// TIA Portal V17 export
// export: Created 2022-03-12T16:05:35.2903502Z, ExportSetting WithDefaults, DisplayName Totally Integrated Automation Portal, DisplayVersion V17, DisplayName TIA Portal Openness, DisplayVersion V17, DisplayName TIA Portal Version Control Interface, DisplayVersion V17, DisplayName STEP 7 Professional, DisplayVersion V17, DisplayName STEP 7 Safety, DisplayVersion V17, DisplayName WinCC Advanced / Unified PC, DisplayVersion V17
TYPE "typeLPMLV30_Diagnostics"
TITLE = typeLPMLV30_Diagnostics
// Support: tech.team.motioncontrol@siemens.com 
// Fax: +49 (0) 9131/98-1297
// stored: IsFailsafeCompliant false
   STRUCT
      bufferIndex : Int := -1;   // Index of actual buffer entry
      buffer { S7_SetPoint := 'True'} : Array[0.."LPMLV30_DIAG_BUFFER_UPPER_LIM"] of "typeLPMLV30_DiagnosticsEntry";   // Diagnostics information buffer
   END_STRUCT;
END_TYPE
